// TIA Portal V16 export
// export: Created 2021-07-06T05:47:27.2187087Z, ExportSetting WithDefaults, DisplayName Totally Integrated Automation Portal, DisplayVersion V16 Update 4, DisplayName TIA Portal Version Control Interface, DisplayVersion V16 Update 2, DisplayName TIA Portal Openness, DisplayVersion V16 Update 4, DisplayName STEP 7 Professional, DisplayVersion V16 Update 4, DisplayName STEP 7 Safety, DisplayVersion V16, DisplayName WinCC Advanced, DisplayVersion V16 Update 4
FUNCTION "ProcessSensor" : Void   // FC1, F_FBD
{ S7_Optimized_Access := 'TRUE' }
VERSION : 0.1
// stored: AutoNumber true, IsIECCheckEnabled false, UDAEnableTagReadback false
   VAR_INPUT
      ctrl : "SensorControl";
   END_VAR
   VAR_OUTPUT
      state : "SensorState";
      safe : Bool;
   END_VAR
BEGIN

REGION Network 1
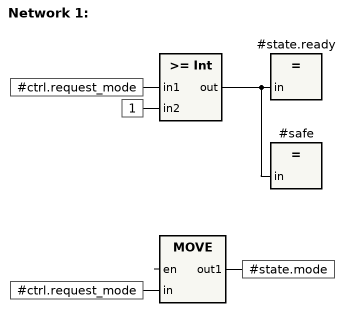
   #state.ready := #ctrl.request_mode >= 1;
   #safe := #state.ready;
   #state.mode := #ctrl.request_mode;
END_REGION
END_FUNCTION
